SUBAPPLICATION Uebung_080 (* Beispiel für E_CTU *)
  (* Standard: 61499-2; Description: Beispiel für E_CTU Aufwärts zählen UAO Curriculum Module 3 - The IEC 61499 Standard, Seite 92 *)
  (* Version 1.0, 2023-10-23, franz *)
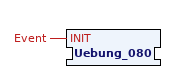
  EVENT_INPUT
    INIT;
  END_EVENT
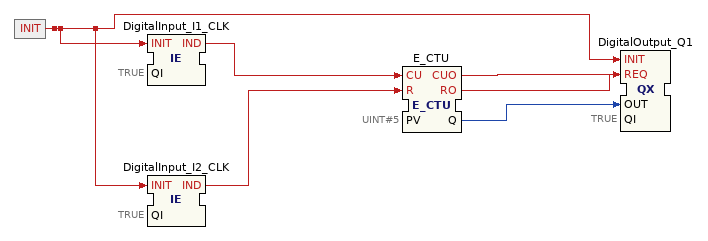
  FBS
    DigitalOutput_Q1 : QX(QI := TRUE);
    DigitalInput_I1_CLK : IE(QI := TRUE);
    E_CTU : E_CTU(PV := UINT#5);
    DigitalInput_I2_CLK : IE(QI := TRUE);
  END_FBS
  EVENT_CONNECTIONS
    INIT TO DigitalInput_I1_CLK.INIT;
    INIT TO DigitalOutput_Q1.INIT;
    DigitalInput_I1_CLK.IND TO E_CTU.CU;
    E_CTU.CUO TO DigitalOutput_Q1.REQ;
    E_CTU.RO TO DigitalOutput_Q1.REQ;
    INIT TO DigitalInput_I2_CLK.INIT;
    DigitalInput_I2_CLK.IND TO E_CTU.R;
  END_CONNECTIONS
  DATA_CONNECTIONS
    E_CTU.Q TO DigitalOutput_Q1.OUT;
  END_CONNECTIONS
END_SUBAPPLICATION
